// TwinCAT 3 PLC project Hausaufgaben_Flankenauswertung
// ProgramVersion: 3.1.4026.16
// libraries:
//   Tc2_Standard, * (Beckhoff Automation GmbH)
//   Tc2_System, * (Beckhoff Automation GmbH)
// project tree:
//   / PlcTask.TcTTO
//   POUs/ FB_DataSim.TcPOU, FB_DatenDurchschnitt.TcPOU, FB_DataStack.TcPOU, FB_Mx_FN_Reset.TcPOU, FB_Mx_FP_Reset.TcPOU, FC_Durchschnitt.TcPOU, FC_GetMaxValue.TcPOU, FC_GetMinValue.TcPOU, R_TRIG.TcPOU, MAIN.TcPOU, F_TRIG.TcPOU
// (motion and I/O tree: see PLC project hausaufgaben_flipflop)
// real-time tasks:
//   TASK PlcTask: cycle T#10ms, priority 20, ADS port 350
//   TASK PlcTask1: cycle T#10ms, priority 21, ADS port 351
//   TASK PlcTask2: cycle T#10ms, priority 22, ADS port 352
//   TASK PlcTask3: cycle T#10ms, priority 23, ADS port 353
//   TASK PlcTask4: cycle T#10ms, priority 24, ADS port 354

CONFIGURATION Hausaufgaben_Flankenauswertung
    RESOURCE PLC ON TwinCAT3
        TASK PlcTask(INTERVAL := T#10ms, PRIORITY := 22);
        PROGRAM MAIN WITH PlcTask : MAIN;
    END_RESOURCE
END_CONFIGURATION

// ---- POUs/MAIN.TcPOU
PROGRAM MAIN
VAR
	Postivie_Flankenerkennung: R_TRIG;				// Instanzierung des R_TRIG-FB's
	ix_Reset: BOOL;									// Abzufragendes Eingangssignal für beide Trigger
	Mx_FP_Reset: BOOL;								// Ausgangsvariable des R_TRIG
	Mx_lmp_Reset_R: BOOL;							// Merker um das Rücksetzten im PG abzufragen
	Negative_Flankenerkennung: F_TRIG;				// Instanzierung des F_TRIG-FB's
	Mx_FN_Reset: BOOL;								// Ausgangsvariable des F_TRIG
	Mx_lmp_Reset_F: BOOL;							// Merker um das Rücksetzten im PG abzufragen
	DatenDurchschnitt: FB_DatenDurchschnitt;
	DatenSim: FB_DataStack;
	DataSim: FB_DataSim;
	DataStack: FB_DataStack;
END_VAR

Postivie_Flankenerkennung(CLK:= ix_Reset);			// Aufruf des R-TRIG
Mx_FP_Reset:= Postivie_Flankenerkennung.Q;			// Zuweisung der Variablen
Mx_lmp_Reset_R:= Mx_FP_Reset;						//

Negative_Flankenerkennung(CLK:= ix_Reset);			// Aufruf des F_TRIG
Mx_FN_Reset:= Negative_Flankenerkennung.Q;			// Zuweisung der Variablen
Mx_lmp_Reset_F:= Mx_FN_Reset;						//

DatenDurchschnitt();
DataSim();

END_PROGRAM

// ---- POUs/R_TRIG.TcPOU
FUNCTION_BLOCK R_TRIG				// FB zur positive Flankenauswertung (Rising Trigger)
VAR_INPUT
	CLK: BOOL;						// Eingangssignal
END_VAR
VAR_OUTPUT
	Q: BOOL;						// Ausgangssignal
END_VAR
VAR
	Last_CLK: BOOL;					// Zwischenspeicher des letzten Zustandes
END_VAR

Q:= CLK AND NOT Last_CLK;
Last_CLK := CLK;

END_FUNCTION_BLOCK

// ---- POUs/F_TRIG.TcPOU
FUNCTION_BLOCK F_TRIG				// FB zur negativen Flankenauswertung (Falling Trigger)		
VAR_INPUT
	CLK: BOOL;						// Zu detektierendes Eingangssignal
END_VAR
VAR_OUTPUT
	Q: BOOL;						// Ausgangssignal wenn Flanke erkannt
END_VAR
VAR
	LastCLK: BOOL;					// Zwischenspeicher des letzten Zustandes von CLK
END_VAR

Q:= NOT CLK AND LastCLK;
LastCLK:= CLK;

END_FUNCTION_BLOCK

// ---- POUs/FB_DatenDurchschnitt.TcPOU
FUNCTION_BLOCK FB_DatenDurchschnitt
VAR_INPUT
END_VAR
VAR_OUTPUT
END_VAR
VAR
	vqr_Durchschnitt: REAL;
	Wert1: INT := 10;
	Wert2: INT := 10;
	Wert3: INT := 10;
END_VAR

vqr_Durchschnitt := FC_Durchschnitt(vii_Wert_1 := Wert1 , vii_Wert_2 :=  Wert2, vii_Wert_3 := Wert3);

END_FUNCTION_BLOCK

// ---- POUs/FC_Durchschnitt.TcPOU
FUNCTION FC_Durchschnitt : REAL				// FC um Durchschnitt zu berechnen
VAR_INPUT
	vii_Wert_1 : INT;						// Einganswert 1
	vii_Wert_2 : INT;						// Einganswert 2
	vii_Wert_3 : INT;						// Einganswert 3
END_VAR
VAR_OUTPUT
END_VAR
VAR
END_VAR

 FC_Durchschnitt := INT_TO_REAL(vii_Wert_1 + vii_Wert_2 + vii_Wert_3) / 3;			// Addition der 3 Werte anschliessend :3 um den Schnitt zu erhalten
// Funktion kann, mit der Übergabe 3er Werte, aus einem beliebigen FB aufgerufen werden. Auch als Multiinstanz aufrufbar

END_FUNCTION

// ---- POUs/FB_DataStack.TcPOU
FUNCTION_BLOCK FB_DataStack
VAR_INPUT
	rValue: REAL;
END_VAR
VAR_OUTPUT
	rAverage: REAL;
END_VAR
VAR
	DataStack: ARRAY[0..100] OF REAL;
	iInPos: INT := 1;
	i: INT;
	rTotal: REAL;
	rMaxValue: REAL;
	rMinValue: REAL;
END_VAR

DataStack[iInPos] := rValue;				//aktueller Wert zur Abspeicherung

IF iInPos >= 100 THEN						//Speicherpositionsbedingung im Array
	iInPos := 1;							//
ELSE 										//
	iInPos := iInPos +1;					//
END_IF										//							

rTotal := 0;								//Initialisierung Gesamtwert
FOR i := 1 TO 100 BY 1 DO					
    rTotal := rTotal + DataStack[i];		//Berechnung Summe aller gespeicherten Werte
END_FOR
rAverage := rTotal / 100;					//Durchschnittsberechnung (Mittelwert je Wert)

rMaxValue := FC_GetMaxValue(MaxValue := DataStack);
rMinValue := FC_GetMinValue(MinValue := DataStack);

END_FUNCTION_BLOCK

// ---- POUs/FC_GetMaxValue.TcPOU
FUNCTION FC_GetMaxValue : REAL
VAR_INPUT
END_VAR
VAR
	iCurrentPos: INT;
END_VAR
VAR_IN_OUT
	MaxValue: ARRAY[0..100] OF REAL;
END_VAR

MaxValue[0] := 0;

FOR iCurrentPos := 1 TO 100 BY 1 DO
	IF MaxValue[iCurrentPos] > MaxValue[0] THEN
		MaxValue[0] := MaxValue[iCurrentPos];
	END_IF
END_FOR

FC_GetMaxValue := MaxValue[0];

END_FUNCTION

// ---- POUs/FC_GetMinValue.TcPOU
FUNCTION FC_GetMinValue : REAL
VAR_INPUT
END_VAR
VAR
	iCurrentPos: INT;
END_VAR
VAR_IN_OUT
	MinValue: ARRAY[0..100] OF REAL;
END_VAR

MinValue[0] := 3.402823E+38;

FOR iCurrentPos := 1 TO 100 BY 1 DO
	IF MinValue[iCurrentPos] < MinValue[0] THEN
		MinValue[0] := MinValue[iCurrentPos];
	END_IF
END_FOR

FC_GetMinValue := MinValue[0];

END_FUNCTION

// ---- POUs/FB_DataSim.TcPOU
FUNCTION_BLOCK FB_DataSim
VAR_INPUT
END_VAR
VAR_OUTPUT
	rValue: REAL := 1.0000;
END_VAR
VAR
	CountTimer: TON;
	RisingEdge: R_TRIG;
	DataStack: FB_DataStack;
END_VAR

CountTimer(IN := TRUE, PT := T#100MS);
RisingEdge(CLK:= CountTimer.Q);

IF RisingEdge.Q AND rValue < 10000 THEN
	rValue := rValue * LREAL_TO_REAL(PI);
	DataStack(rValue := rValue);
ELSIF RisingEdge.Q AND rValue > 10000 THEN
	rValue := (rValue /100) * 1.75;
	DataStack(rValue := rValue);
END_IF

IF CountTimer.Q THEN
	CountTimer(IN := FALSE);
	CountTimer(IN := TRUE);
END_IF

END_FUNCTION_BLOCK

// ---- POUs/FB_Mx_FN_Reset.TcPOU
FUNCTION_BLOCK FB_Mx_FN_Reset			// FB zum erkennen einer fallender Flanke
VAR_INPUT
	Ix_Reset: BOOL;						// Abzufragendes Signal
END_VAR
VAR_OUTPUT
END_VAR
VAR
	Mx_lmp_Reset: BOOL;					// Ausgang für 1 Zyklus aktiv wenn negative Flanke erkannt  
	last_CLK: BOOL;						// Zwischenspeicher des letzten Zustandes des Eingangssignal
END_VAR

Mx_lmp_Reset := NOT Ix_Reset AND last_CLK;		// Ausgang schaltet für 1 Zyklus auf TRUE wenn Bedingung erfüllt, ansonsten bleibt er FALSE	
last_CLK := Ix_Reset;							// Zwischenspeicher des letzten Zustandes des abzufragenden Signals (Ix_Reset)

//Auch Möglich umzusetzten mit IF, ELSE:

IF last_CLK AND NOT Ix_Reset THEN				// Wenn Bedingung einer fallenden Flanke erfüllt
	Mx_lmp_Reset := TRUE;						// Ausgang schaltet für 1 Zyklus auf TRUE
ELSE 
	Mx_lmp_Reset := FALSE;						// Wenn Bedingung einer fallenden Flanke nicht erfüllt bleibt Ausgang FALSE
END_IF
last_CLK := Ix_Reset;							// Zwischenspeicher des letzten Zustandes des abzufragenden Signals (Ix_Reset)

END_FUNCTION_BLOCK

// ---- POUs/FB_Mx_FP_Reset.TcPOU
FUNCTION_BLOCK FB_Mx_FP_Reset			// FB zum erkennen einer steigender Flanke
VAR_INPUT
	Ix_Reset: BOOL;						// Abzufragendes Signal
END_VAR
VAR_OUTPUT
END_VAR
VAR
	Mx_lmp_Reset: BOOL;					// Ausgang für 1 Zyklus aktiv wenn negativepositive Flanke erkannt
	last_CLK: BOOL;						// Zwischenspeicher des letzten Zustandes des Eingangssignal
END_VAR

Mx_lmp_Reset:= Ix_Reset AND NOT last_CLK;		// Ausgang schaltet für 1 Zyklus auf TRUE wenn Bedingung erfüllt, ansonsten bleibt er FALSE	
last_CLK:= Ix_Reset;							// Zwischenspeicher des letzten Zustandes des abzufragenden Signals (Ix_Reset)

//Auch Möglich umzusetzten mit IF, ELSE:

IF NOT last_CLK AND Ix_Reset THEN				// Wenn Bedingung einer steigender Flanke erfüllt
	Mx_lmp_Reset := TRUE;						// Ausgang schaltet für 1 Zyklus auf TRUE
ELSE 
	Mx_lmp_Reset := FALSE;						// Wenn Bedingung einer steigender Flanke nicht erfüllt bleibt Ausgang FALSE
END_IF
last_CLK := Ix_Reset;							// Zwischenspeicher des letzten Zustandes des abzufragenden Signals (Ix_Reset)

END_FUNCTION_BLOCK
